{attribute addProperty BoxType "KL9900-0063"}
{attribute addProperty Id "Channel_1Channel_E28253B100"}
{attribute addProperty CRC "1624091552"}
{attribute addProperty SizeInBites "0"}
{attribute addProperty SizeInBytes "0"}
TYPE KL_60CDABA0 :
STRUCT
	{attribute addProperty Name "Channel_1"}
	Channel_1 : Channel_E28253B1;
END_STRUCT
END_TYPE

(* stored: Version 1.2.0.0, ProductVersion 3.1.4024.9
   DUT KL_60CDABA0: Id {a6ebeba7-8672-4912-8b99-335de002f3f3} *)
